(*
Standard way to set up events to be tied to other parts of the project. might make an interface
*)

FUNCTION_BLOCK FB_DiscreteEvents
VAR_INPUT
END_VAR
VAR_OUTPUT
END_VAR
VAR
END_VAR

METHOD FB_init : BOOL
VAR_INPUT
	bInitRetains : BOOL; // if TRUE, the retain variables are initialized (warm start / cold start)
	bInCopyCode : BOOL;  // if TRUE, the instance afterwards gets moved into the copy code (online change)
	eventName : STRING;
	evemtID : DINT;
END_VAR
END_METHOD

METHOD PUBLIC ABSTRACT M_Execute : HRESULT
VAR_INPUT
	lastResult : HResult;
END_VAR
END_METHOD

PROPERTY PUBLIC P_EventId : Dint
GET
END_GET
SET
END_SET
END_PROPERTY

PROPERTY PUBLIC P_EventName : String
GET
END_GET
END_PROPERTY

END_FUNCTION_BLOCK

(* stored: Version 1.1.0.1, ProductVersion 3.1.4024.12
   POU FB_DiscreteEvents: Id {a9950c77-75c4-4565-9d6a-64f0c0ce1cfe}, SpecialFunc None
   Method FB_init: Id {71612a4f-f6aa-4e09-89dc-467927c53386}
   Method M_Execute: Id {1fd5e78f-7de2-40f0-8ed2-a85a6dac936a}
   Property P_EventId: Id {cf51e756-b2bf-4a32-9949-f15b5e95182a}
   Get Get: Id {f62c00b6-2218-4e2c-870d-5cacf6328e6d}
   Set Set: Id {6ff57742-0e5d-4401-a5e2-bf854e8a9974}
   Property P_EventName: Id {c298ca1a-b765-48f4-a6ad-9e9372811d6e}
   Get Get: Id {21c550db-b1f3-4dcb-aefa-7bb3ab289d89} *)
